// TIA Portal V17 export
// export: Created 2023-12-22T15:05:28.2754194Z, ExportSetting WithDefaults, DisplayName Totally Integrated Automation Portal, DisplayVersion V17, DisplayName TIA Portal Openness, DisplayVersion V17, DisplayName TIA Portal Version Control Interface, DisplayVersion V17, DisplayName STEP 7 Professional, DisplayVersion V17, DisplayName STEP 7 Safety, DisplayVersion V17, DisplayName WinCC Advanced, DisplayVersion V17
FUNCTION_BLOCK "AIx"   // FB220, LAD
{ S7_Optimized_Access := 'FALSE' }
VERSION : 0.1
// Signal - PIW код сигнала от датчика
// pulse - частота алгоритма фильтрации
// Result - результат обработки сигнала, формат Real
// stored: AutoNumber false, IsIECCheckEnabled false, SetENOAutomatically false, UDAEnableTagReadback false
   VAR DB_SPECIFIC
      Time_DTL { S7_SetPoint := 'True'} : DTL;
   END_VAR
   VAR_TEMP   // added for the SCL form of the ladder/FBD networks
      _w1 : Bool;
   END_VAR
BEGIN

REGION Network 1: Датчик уровня
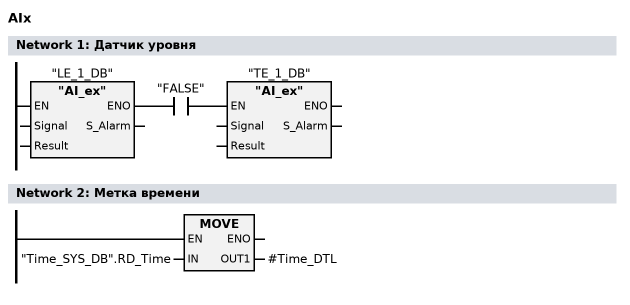
   RUNG wire#powerrail
      "LE_1_DB"(Signal :=, Result :=, S_Alarm =>)
      Contact( "FALSE" )
      "TE_1_DB"(Signal :=, Result :=, S_Alarm =>)
   END_RUNG
   // the same network as SCL:
   "LE_1_DB"(ENO => #_w1);   // "AI_ex"
   IF #_w1 AND "FALSE" THEN
       "TE_1_DB"();   // "AI_ex"
   END_IF;
END_REGION

REGION Network 2: Метка времени
   RUNG wire#powerrail
      Move(in := "Time_SYS_DB".RD_Time, out1 => #Time_DTL)
   END_RUNG
   // the same network as SCL:
   #Time_DTL := "Time_SYS_DB".RD_Time;
END_REGION
END_FUNCTION_BLOCK
